FUNCTION_BLOCK FB_OM_SemiAuto
VAR_INPUT
END_VAR
VAR_OUTPUT
	eCurrentState : E_MachineState := E_MachineState.MACHINESTATE_Idle;
END_VAR
VAR
	nCalls	: UINT;
END_VAR

nCalls := nCalls + 1;

METHOD M_ResetError
VAR_INPUT
END_VAR
END_METHOD

END_FUNCTION_BLOCK

(* stored: Version 1.1.0.1, ProductVersion 3.1.4022.7
   POU FB_OM_SemiAuto: Id {46128769-d126-4300-8b7c-225de175655d}, SpecialFunc None
   Method M_ResetError: Id {dd4081f0-8c07-440b-9fe8-50f498f04c33} *)
